{attribute 'qualified_only'}
VAR_GLOBAL CONSTANT
	COMMAND_QUEUE_BUFFER_SIZE :UDINT := 64; // Queue size for database insert command.
	DATA_BUFFER_SIZE	:UDINT := 500; // Data buffer size
	MAX_COLUMN_NUM		: UDINT := 50;
END_VAR

(* stored: Version 1.1.0.1, ProductVersion 3.1.4024.12
   GVL DBLibParam: Id {56321c42-7c93-46e8-98ed-6ddc16ce704e}, ParameterList True *)
